// TIA Portal V21 export
FUNCTION "FC_Modelo" : Void   // FC210, LAD
{ S7_Optimized_Access := 'TRUE' }
VERSION : 0.1
// stored: AutoNumber true, IsIECCheckEnabled false, SetENOAutomatically false, UDAEnableTagReadback false
BEGIN

REGION Network 1: Word de Alarmes: MODELO
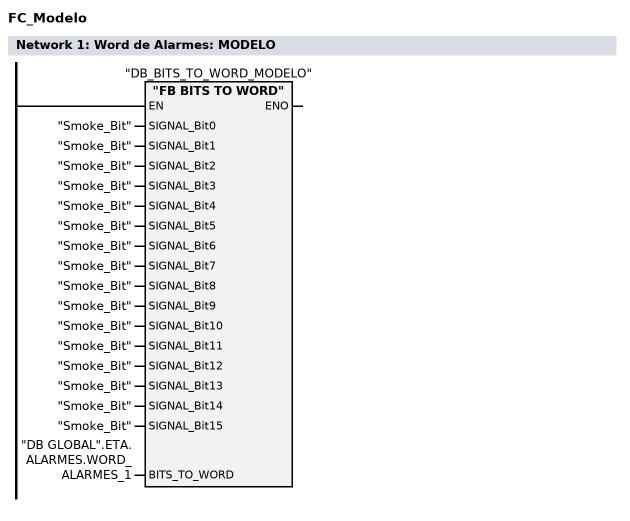
   RUNG wire#powerrail
      "DB_BITS_TO_WORD_MODELO"(SIGNAL_Bit0 := "Smoke_Bit", SIGNAL_Bit1 := "Smoke_Bit", SIGNAL_Bit2 := "Smoke_Bit", SIGNAL_Bit3 := "Smoke_Bit", SIGNAL_Bit4 := "Smoke_Bit", SIGNAL_Bit5 := "Smoke_Bit", SIGNAL_Bit6 := "Smoke_Bit", SIGNAL_Bit7 := "Smoke_Bit", SIGNAL_Bit8 := "Smoke_Bit", SIGNAL_Bit9 := "Smoke_Bit", SIGNAL_Bit10 := "Smoke_Bit", SIGNAL_Bit11 := "Smoke_Bit", SIGNAL_Bit12 := "Smoke_Bit", SIGNAL_Bit13 := "Smoke_Bit", SIGNAL_Bit14 := "Smoke_Bit", SIGNAL_Bit15 := "Smoke_Bit", BITS_TO_WORD := "DB GLOBAL".ETA.ALARMES.WORD_ALARMES_1)
   END_RUNG
   // the same network as SCL:
   "DB_BITS_TO_WORD_MODELO"(SIGNAL_Bit0 := "Smoke_Bit",   // "FB BITS TO WORD"
                           SIGNAL_Bit1 := "Smoke_Bit",
                           SIGNAL_Bit2 := "Smoke_Bit",
                           SIGNAL_Bit3 := "Smoke_Bit",
                           SIGNAL_Bit4 := "Smoke_Bit",
                           SIGNAL_Bit5 := "Smoke_Bit",
                           SIGNAL_Bit6 := "Smoke_Bit",
                           SIGNAL_Bit7 := "Smoke_Bit",
                           SIGNAL_Bit8 := "Smoke_Bit",
                           SIGNAL_Bit9 := "Smoke_Bit",
                           SIGNAL_Bit10 := "Smoke_Bit",
                           SIGNAL_Bit11 := "Smoke_Bit",
                           SIGNAL_Bit12 := "Smoke_Bit",
                           SIGNAL_Bit13 := "Smoke_Bit",
                           SIGNAL_Bit14 := "Smoke_Bit",
                           SIGNAL_Bit15 := "Smoke_Bit",
                           BITS_TO_WORD := "DB GLOBAL".ETA.ALARMES.WORD_ALARMES_1);
END_REGION
END_FUNCTION
